FUNCTION_BLOCK FB_BINARY_SWITCH_SENS IMPLEMENTS  I_BINARY_SWITCH_SENS
VAR_INPUT
END_VAR
VAR_OUTPUT
END_VAR
VAR
		
	itfOpMode:										I_OP_MODE;
	{attribute 'instance-path'} 
    {attribute 'noinit'} 
	strInstancePath:								STRING;
	strFullObjectPath:								STRING;
	stEvent:										ST_EVENT;
	bAck:											BOOL;
	
	bSwitch 										AT %I*: BOOL;
	bNC:											BOOL;
	fbEventLogger:									FB_TcEventLogger;
	                                				
	strSymName:										STRING;
	iStepCase:										INT;
	strMessage:										STRING;
	bSensingON:										BOOL;
END_VAR

strFullObjectPath:=F_CreateIdString(THIS^);


stEvent.bEventActive:=FALSE;
IF THIS^.bSensingON AND P_Active THEN
	fbEventLogger.GetAlarm(eventClass:= TC_EVENT_CLASSES.TcSystemEventClass,
							nEventID:=1,
							ipSourceInfo:=TRUE,
							fbAlarm:=TRUE);
END_IF



//Überwachung Eingang
CASE iStepCase OF
	
	0://SENSING Deaktiviert
	
	
	1://SENSING Aktiviert
		
		
	
	
	re
END_CASE

METHOD FB_init : BOOL
VAR_INPUT
	bInitRetains : BOOL; // if TRUE, the retain variables are initialized (warm start / cold start)
	bInCopyCode : BOOL;  // if TRUE, the instance afterwards gets moved into the copy code (online change)
	itfOpMode:			I_OP_MODE;
	bInNC: 				BOOL;///NC:=true; NO:= false
	strMessage:			STRING;
	bSensingON:			BOOL;
END_VAR
THIS^.itfOpMode:=	itfOpMode;
THIS^.bNC:=			bInNC;
THIS^.strMessage:=	strMessage;
THIS^.bSensingON:=	bSensingON;
END_METHOD

(*=== Method: M_Run  ============================================

 @brief: Here is the global code (Timer, Event, Flange,...)*)
METHOD M_Run
END_METHOD

METHOD M_START_SENS : BOOL
VAR_INPUT
	bState	: BOOL;
	tDelay	: TIME;
	eEventType	: GenLib.ENUM_EVENT_TYPE;
END_VAR
IF THIS^.iStepCase=0 THEN
	THIS^.iStepCase:=1;
END_IF
END_METHOD

METHOD M_STOP_SENS : BOOL
END_METHOD

PROPERTY P_Active : BOOL
GET
IF bNC THEN
	P_ACTIVE:= NOT bSwitch;
ELSE
	P_ACTIVE:= bSwitch;
END_IF
END_GET
END_PROPERTY

(*=== Property: P_Event  ============================================

 @param [set]: 	Set the Structure "ST_EVENT" from another Object
 @param [get]: 	Return the Structure "ST_EVENT", it contains the actual 
					event of the Object *)
PROPERTY P_Event : GenLib.ST_EVENT
GET
P_Event:=stEvent;
END_GET
SET
stEvent:=P_Event;
END_SET
END_PROPERTY

(*=== Property: P_FullObjectPath  ============================================

 @param [set]: 	Set the Object Path (Clear String of Object)
 @param [get]: 	Return the Objectpath *)
PROPERTY P_FullObjectPath : STRING
GET
P_FullObjectPath:= THIS^.strFullObjectPath;
END_GET
SET
END_SET
END_PROPERTY

(*=== Property: P_Global_Ack  ============================================

 @param [set]: 	Set the Bit for Ack from another Object
 @param [get]: 	Return the state of Ack Bit*)
PROPERTY P_Global_Ack : BOOL
GET
P_Global_Ack:=THIS^.bAck;
END_GET
SET
THIS^.bAck:=P_Global_Ack;
END_SET
END_PROPERTY

{warning 'Eigenschaftenimplementierung hinzufügen'}
(*=== Property: P_GlobalID  ============================================

 @param [set]: 	-
 @param [get]: 	Return the string of instance path*)
PROPERTY P_GlobalID : STRING
GET
P_GlobalID:= THIS^.strInstancePath;
END_GET
END_PROPERTY

PROPERTY P_No_Nc : BOOL
GET
P_No_Nc:= not THIS^.bNC;
END_GET
END_PROPERTY

PROPERTY P_On : BOOL
GET
P_ON:= bSwitch;
END_GET
END_PROPERTY

PROPERTY P_STATE_SENS : BOOL
GET
END_GET
END_PROPERTY

END_FUNCTION_BLOCK

(* stored: Version 1.1.0.1, ProductVersion 3.1.4024.12
   POU FB_BINARY_SWITCH_SENS: Id {a6e1280c-511a-4b66-8a42-e759c894cb17}, SpecialFunc None
   Method FB_init: Id {612c5594-60d2-4cb6-ad38-deb99a021cb6}
   Method M_Run: Id {dbfa0a1d-8709-477b-a87a-771fd441aa29}
   Method M_START_SENS: Id {c67b2c3b-ff44-4f79-8aa2-87e9ad17816b}
   Method M_STOP_SENS: Id {1d7a551c-f96b-46ea-a4d4-92b6e76e4cc0}
   Property P_Active: Id {a021e4ad-1a58-49c3-b16c-28454108738c}
   Get Get: Id {c40f50bd-8865-4e24-b443-d1f919e081ab}
   Property P_Event: Id {9a927b0f-ca3a-490c-a56f-436b387c1189}
   Get Get: Id {63f12604-7ba2-4aab-bf7c-d68b2012bcd4}
   Set Set: Id {08ab960d-81bd-47bb-949e-2fd6768e993f}
   Property P_FullObjectPath: Id {1e100d33-612b-4f55-9fa3-af1b40d98813}
   Get Get: Id {211439c7-68ed-4cbc-b681-b0ee6558f078}
   Set Set: Id {190220e9-b6e4-479e-a673-4b203898fa96}
   Property P_Global_Ack: Id {8d4bf222-219f-4041-abbe-1b72a2d51931}
   Get Get: Id {a4e86b95-d3e7-4615-a8e4-73141355307a}
   Set Set: Id {112b517a-163e-4922-9fa8-e9137764a4df}
   Property P_GlobalID: Id {c57749aa-b2d3-4aab-8473-150967d2c379}
   Get Get: Id {96096b9d-3fba-46f1-aa7a-2b14654d007e}
   Property P_No_Nc: Id {81e8d3b9-46ac-4b83-9d73-d7de80949cba}
   Get Get: Id {56b72e5a-df32-4626-bab0-fa73d42af897}
   Property P_On: Id {dc8596ac-a35e-4a8f-83aa-e539b0b3da8f}
   Get Get: Id {d75cb3a6-0374-4fe2-a480-e8d5d92c8f58}
   Property P_STATE_SENS: Id {95e03ebd-e4c3-4c60-b996-477980271428}
   Get Get: Id {25a60d37-381d-49c2-9721-ccf49babf667} *)
